// TIA Portal V19 export
VAR_GLOBAL   // PLC tag table "Unit3_Input"
END_VAR
